FUNCTION_BLOCK ButtonsPanel_HMI (* Service Interface Function Block Type *)
  (* Standard: 61499-2 *)
  (* Version 0.0, 7/13/2016, Andrei, nxtControl GmbH, template *)
  PACKAGE Main;
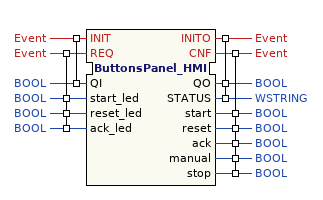
  EVENT_INPUT
    INIT WITH QI;
    REQ WITH start_led, reset_led, ack_led;
  END_EVENT
  EVENT_OUTPUT
    INITO WITH QO, STATUS;
    CNF WITH start, reset, ack, manual, stop;
  END_EVENT
  VAR_INPUT
    QI : BOOL;
    start_led : BOOL;
    reset_led : BOOL;
    ack_led : BOOL;
  END_VAR
  VAR_OUTPUT
    QO : BOOL; (* Event Output Qualifier *)
    STATUS : WSTRING; (* Service Status *)
    start : BOOL;
    reset : BOOL;
    ack : BOOL;
    manual : BOOL;
    stop : BOOL;
  END_VAR
END_FUNCTION_BLOCK
